# EPICS substitutions: ADnED/example/exampleApp/Db/example.substitutions
file ADnED.template
{
pattern {P, ADNED, PORT, ADDR, TIMEOUT, TOFSIZE, ADNED_PORT, TOF1SIZE, TOF2SIZE, TOF3SIZE, TOF4SIZE, DET1SIZE, DET2SIZE, DET3SIZE, DET4SIZE, DET1X, DET2X, DET3X, DET4X, DET1Y, DET2Y, DET3Y, DET4Y}
	{BL99:Det:, N1:, N1, 0, 5, 160000, N1,               1600, 1600, 16000, 16000,         1024,     1024,     5120,    163840,    32,    32,    160,  160,     32,    32,    32,     32}
	{BL99:Det:, M1:, M1, 0, 5, 160000, M1,               160000, 160000, 160000, 160000,         1024,     1024,     0,        0,        32,    32,    0,     0,     32,    32,    0,     0}
}

file save_restoreStatus.db
{
pattern {P}
        {BL99:CS:Det:ADnED:}
}

file ioc_sns.db
{
pattern {IOCNAME}
        {BL99:CS:Det:ADnED}
}
